FUNCTION_BLOCK FB_MachineState IMPLEMENTS I_MachineStateBase
(*************************************************************************************************)
(*  FILENAME:    FB_MachineState                                                                 *)
(*  PROJECT:     CALMAR PUPLC                                                                    *)
(*  COPYRIGHT:   All rights reserved (c) Polytype AG, Fribourg/Switzerland (2020)                *)
(*  ENVIRONMENT: TwinCAT PLC                                                                     *)
(*  VERSION:     <version>                                                                       *)
(*************************************************************************************************)
(*  DESCRIPTION:                                                                   <description> *)
(*    add description                                                                            *)
(*                                                                                </description> *)
(*************************************************************************************************)

VAR_INPUT
  bI_SafetyOk                     : BOOL;  (*Safety ok for movement*)
  bI_MachineReady                 : BOOL;  (*Machine ready*)
END_VAR

PROPERTY pMachineReady : BOOL
GET
pMachineReady := bI_MachineReady;
END_GET
END_PROPERTY

PROPERTY pSafetyOk : BOOL
GET
pSafetyOk := bI_SafetyOk;
END_GET
END_PROPERTY

END_FUNCTION_BLOCK

(* stored: Version 1.1.0.1, ProductVersion 3.1.4024.11
   POU FB_MachineState: Id {99306a14-ffa2-4e55-ab7a-3166624cfb8a}, SpecialFunc None
   Property pMachineReady: Id {916e6e73-8c20-4a41-848d-0dec9b17ccfb}
   Get Get: Id {b5547524-c2ed-4117-b5b3-a9eb5cc3fce1}
   Property pSafetyOk: Id {db974116-5989-4c02-9d25-9a14db407c1f}
   Get Get: Id {45c11563-1e50-4f32-bb3e-e8f5d62ab6ae} *)
